{attribute 'GeneratedUsingTerminal: EL2212-0000-0020'}
{attribute addProperty BoxType "EL2212-0000-0020"}
{attribute addProperty Id "ControlAT %Q*Control_87176C1F4"}
{attribute addProperty CRC "3868395073"}
{attribute addProperty Size "4"}
TYPE DOX_Control_Channel_E6930641 :
STRUCT
	{attribute addProperty Name "Control"}
	Control AT %Q* : Control_87176C1F;
END_STRUCT
END_TYPE

(* stored: Version 1.2.0.0, ProductVersion 3.1.4024.9
   DUT DOX_Control_Channel_E6930641: Id {8a52784a-7de6-4ef8-910a-6a37e12f9a18} *)
